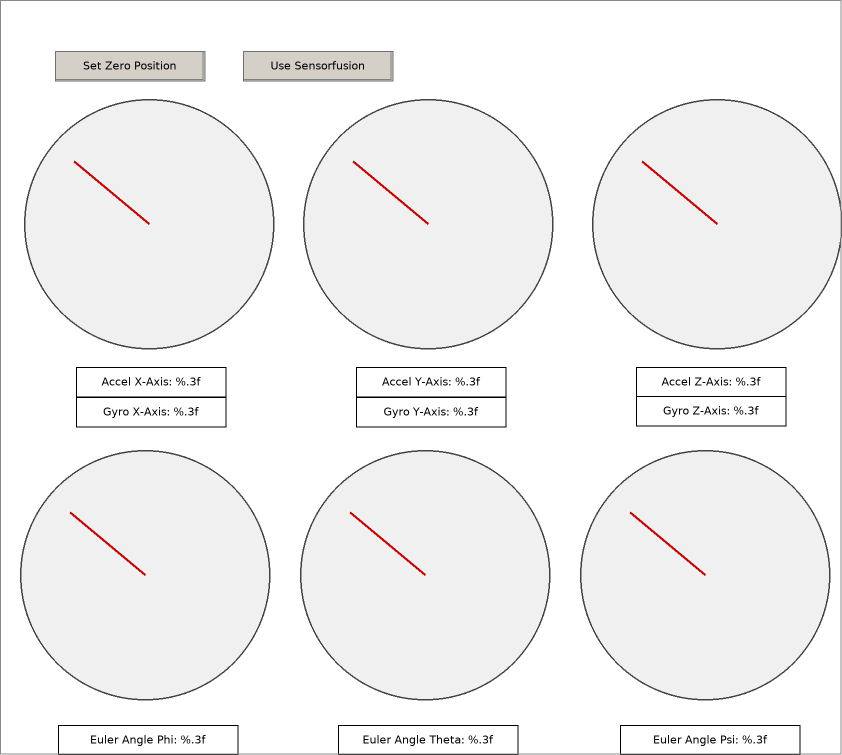
VISUALIZATION Visualization_Mahony  // 842x755
    Meter360 (24,99 250x250), value: MAIN.a_fAccAxis[0], style: Meter-Meter360-Gray, scale format: %.2f, scale -2..2
        p518627256: °
    Rectangle (76,367 150x30), "Accel X-Axis: %.3f", text variable: MAIN.a_fAccAxis[0]
    Button (55,51 150x30), "Set Zero Position", colour toggle: MAIN.bReady
        p2175578022: 16#FF808080
        p573394764: 16#FF80FF80
        tap MAIN.bReset
    Rectangle (356,367 150x30), "Accel Y-Axis: %.3f", text variable: MAIN.a_fAccAxis[1]
    Rectangle (636,367 150x30), "Accel Z-Axis: %.3f", text variable: MAIN.a_fAccAxis[2]
    Rectangle (76,397 150x30), "Gyro X-Axis: %.3f", text variable: MAIN.a_fGyroAxis[0]
    Rectangle (356,397 150x30), "Gyro Y-Axis: %.3f", text variable: MAIN.a_fGyroAxis[1]
    Rectangle (636,396 150x30), "Gyro Z-Axis: %.3f", text variable: MAIN.a_fGyroAxis[2]
    Button (243,51 150x30), "Use Sensorfusion", colour toggle: MAIN.bUseSensorFusion
        p2175578022: 16#FF808080
        p573394764: 16#FF80FF80
        toggle MAIN.bUseSensorFusion
    Meter360 (303,99 250x250), value: MAIN.a_fAccAxis[1], style: Meter-Meter360-Gray, scale format: %.2f, scale -2..2
        p518627256: °
    Meter360 (592,99 250x250), value: MAIN.a_fAccAxis[2], style: Meter-Meter360-Gray, scale format: %.2f, scale -2..2
        p518627256: °
    Meter360 (20,450 250x250), value: MAIN.fbMahonyFilter.fAngleRoll_deg, style: Meter-Meter360-Gray, scale format: %d, scale -180..180
        p518627256: °
    Meter360 (300,450 250x250), value: MAIN.fbMahonyFilter.fAnglePitch_deg, style: Meter-Meter360-Gray, scale format: %d, scale -180..180
        p518627256: °
    Meter360 (580,450 250x250), value: MAIN.fbMahonyFilter.fAngleYaw_deg, style: Meter-Meter360-Gray, scale format: %d, scale -180..180
        p518627256: °
    Rectangle (58,725 180x30), "Euler Angle Phi: %.3f", text variable: MAIN.fbMahonyFilter.fAngleRoll_deg
    Rectangle (338,725 180x30), "Euler Angle Theta: %.3f", text variable: MAIN.fbMahonyFilter.fAnglePitch_deg
    Rectangle (620,725 180x30), "Euler Angle Psi: %.3f", text variable: MAIN.fbMahonyFilter.fAngleYaw_deg
END_VISUALIZATION

(* stored: Version 1.1.0.1, ProductVersion 3.1.4024.13
   Visu Visualization_Mahony: Id {14891dcb-a45c-4244-9c0c-ac9d79b1bba6} *)
